# B&R Automation Studio project PLC code - cp (part 22)

#### Stack.st
```iecst
ACTION Stack:

	(* UA_MethodCall - call methode *)
	InputArguments_0[0].Name := 'MediaData';
	InputArguments_0[0].Value := '::SimMachFst:NewMediaData_0';
	OutputArguments_0[0].Name := 'Result';
	OutputArguments_0[0].Value := '::SimMachFst:MethodResult_0';
	UA_MethodCall_0(Execute := ExecuteMethodCall_0,
		ConnectionHdl := ConnectionHdl_0,
		MethodHdl := MethodHdl_0,
		Timeout := T#10s,
		InputArguments := InputArguments_0,
		OutputArguments := OutputArguments_0);
	IF NOT UA_MethodCall_0.Busy THEN
		ExecuteMethodCall_0 := FALSE;
		IF UA_MethodCall_0.Done THEN
			NewMediaData_0.rLength := NewMediaData_0.rLength + 1;
		END_IF
		IF UA_MethodCall_0.Error THEN
			NewMediaData_0.rDocLength := NewMediaData_0.rDocLength + 1;
		END_IF
	END_IF

	// Managing the automatic sending. Not sending if enable drying. Sendign Energy then
	IF NOT gThicknessCtrl.status.xNewMediaStackEnabled OR gThicknessCtrl.parameters.Dry.xDryStack THEN
		RETURN;
	END_IF

	IF (gSimMachine.Parameters.Stack.iMediaQuantityToKeepLoaded <= gThicknessCtrl.status.Stack.iNewMediaLoadedL1 + gThicknessCtrl.status.Stack.iNewMediaLoadedL2) THEN
		RETURN;
	END_IF

	// Adding a timer to avoid not working the method
	tonNotCallingMethod_0.IN := NOT UA_MethodCall_0.Busy;
	tonNotCallingMethod_0.PT := t#500ms;
	tonNotCallingMethod_0();
	IF EDGEPOS(tonNotCallingMethod_0.Q) THEN
		ExecuteMethodCall_0 := TRUE;
	END_IF

END_ACTION

ACTION InitialDataForMedia:

	NewMediaData_0.iLine := 1;
	NewMediaData_0.xHasWhite := FALSE;
	NewMediaData_0.rThickness := 3;
	NewMediaData_0.rWidth := 1400;
	NewMediaData_0.rLength := 1000;
	NewMediaData_0.rCrossOffset := 0;
	NewMediaData_0.rDocWidth := 1400;
	NewMediaData_0.rDocLength := 950;
	NewMediaData_0.rDocCrossOffset := 0;
	NewMediaData_0.rDocProcessOffset := 0;

END_ACTION

ACTION PreparingMethodComms:

	ExecuteConnect_0 := TRUE;

	(* UA_Connect - establish connection to OPC UA Server *)
	SessionConnectInfo_0.SecurityMsgMode := UASecurityMsgMode_None;
	SessionConnectInfo_0.SecurityPolicy := UASecurityPolicy_None;
	SessionConnectInfo_0.TransportProfile := UATP_UATcp;
	SessionConnectInfo_0.UserIdentityToken.UserIdentityTokenType := UAUITT_Username;
	SessionConnectInfo_0.UserIdentityToken.TokenParam1 := 'PressCore';
	SessionConnectInfo_0.UserIdentityToken.TokenParam2 := 'h98o76';
	SessionConnectInfo_0.SessionTimeout := T#1m;
	SessionConnectInfo_0.MonitorConnection := T#10s;

	UA_Connect_0(Execute := ExecuteConnect_0,
		ServerEndpointUrl := 'opc.tcp://localhost:4840',
	SessionConnectInfo := SessionConnectInfo_0,
	Timeout := T#10s);
	IF NOT UA_Connect_0.Busy THEN
		ExecuteConnect_0 := FALSE;
		IF UA_Connect_0.Done THEN
			ConnectionHdl_0 := UA_Connect_0.ConnectionHdl;
			////// NEXT
			ExecuteGetnamespaceindex_0 := TRUE;
		END_IF
		IF UA_Connect_0.Error THEN
			ConnectionHdl_0 := 0;
		END_IF
	END_IF

	(* UA_GetNamespaceIndex - read index of required namespace for PVs *)
	UA_GetNamespaceIndex_0(Execute := ExecuteGetnamespaceindex_0,
		ConnectionHdl := ConnectionHdl_0,
		NamespaceUri := 'http://br-automation.com/OpcUa/PLC/PV/',
	Timeout := T#5s);
	IF NOT UA_GetNamespaceIndex_0.Busy THEN
		ExecuteGetnamespaceindex_0 := FALSE;
		IF UA_GetNamespaceIndex_0.Done THEN
			NamespaceIndex_0 := UA_GetNamespaceIndex_0.NamespaceIndex;
			////// NEXT
			ExecuteMethodGetHandle_0 := TRUE;
		END_IF
		IF UA_GetNamespaceIndex_0.Error THEN
			NamespaceIndex_0 := 0;
		END_IF
	END_IF

	(* UA_MethodGetHandle - get a handle for required methode *)
	ObjectNodeID_0.NamespaceIndex := NamespaceIndex_0;
	ObjectNodeID_0.Identifier := '::ThickPos';
	ObjectNodeID_0.IdentifierType := UAIdentifierType_String;
	MethodNodeID_0.NamespaceIndex := NamespaceIndex_0;
	MethodNodeID_0.Identifier := '::ThickPos:LoadNewMedia';
	MethodNodeID_0.IdentifierType := UAIdentifierType_String;
	UA_MethodGetHandle_0(Execute := ExecuteMethodGetHandle_0,
		ConnectionHdl := ConnectionHdl_0,
		ObjectNodeID := ObjectNodeID_0,
		MethodNodeID := MethodNodeID_0,
		Timeout := T#10s);
	IF NOT UA_MethodGetHandle_0.Busy THEN
		ExecuteMethodGetHandle_0 := FALSE;
		IF UA_MethodGetHandle_0.Done THEN
			MethodHdl_0 := UA_MethodGetHandle_0.MethodHdl;
			////// NEXT
			// READY TO COMMUNICATE
		END_IF
		IF UA_MethodGetHandle_0.Error THEN
			MethodHdl_0 := 0;
		END_IF
	END_IF

END_ACTION
```

- Visualisation Logical/Printer/Sim/SimVisu (not shown)

### TestResources.var
```iecst
VAR
	iIndex : UDINT;
	iMax : UDINT;
	rVal : REAL;
END_VAR
```

- Visualisation Logical/Printer/mappView (not shown)

### Library Logical/UnitTest/Libraries/EFIAssert (ANSIC)

#### EFIAssert_ThresholdAssert.h - Threshold: macros
```c
/********************************************************************
 * COPYRIGHT -- Bernecker + Rainer
 ********************************************************************
 * Library: EFIAssert
 * File: EFIAssert_ThresholdAssert.h
 * Author: B+R
 *******************************************************************/

#include <bur/plctypes.h>

#include <bur/plctypes.h>
#include "UnitTest.h"

#ifdef __cplusplus
extern "C"
{
#endif

/* Dummies for smart edit autocompletion.
See below for the real macros used by the compiler  */
#ifdef _SMART_EDIT_DUMMY_
	/* This asserts checks (actual < threshold) */
	BOOL SPLEFI_ASSERT_UPPER_BOUNDARY(DINT threshold, DINT actual);
#endif

/*------------------------------------------------------------*/

/* Prototyping of functions.
These declaration of functions are used by the compiler to check number and type of arguments. */
BOOL splefi_assertUpperBoundary_DINT(const DINT threshold, const DINT actual, unsigned long line, const char *file);

/* Macros used in the test implementation.
The macro passes the location information to the implemented assert. */
#define SPLEFI_ASSERT_UPPER_BOUNDARY(threshold, actual) 	\
	splefi_assertUpperBoundary_DINT(threshold, actual, (unsigned long) __LINE__, __FILE__)

#ifdef __cplusplus
};
#endif
```

#### EFIAssert_REAL_ArrayAsserts.c - Array of REAL: implementation of the assert
```c
/********************************************************************
 * COPYRIGHT -- Bernecker + Rainer
 ********************************************************************
 * Library: EFIAssert
 * File: EFIAssert_REAL_ArrayAsserts.c
 * Author: B+R
 *******************************************************************/

#include <bur/plctypes.h>

#include "asbrstr.h"
#include "EFIAssert_REAL_ArrayAsserts.h"

#define TRUE 1
#define FALSE 0

#define NR_OF_DETAILED_ENTRIES_TO_SHOW 10

/* Tests each REAL in the array for equality in range
Returns true if passed, false otherwise
delta: allowed tolerance (floats are not exact values)
expected: array of expected REAL values
acutal: array of REAL values under test
nrOfEntries: number of entries in array
line: location information
file: location information
*/
BOOL splefi_assertImplRealArrayWithin(const REAL *delta,
                                   const REAL *expected, 	const REAL *actual, const unsigned long nrOfEntries,
                                   unsigned long line, const char *file)
{
	unsigned long i = 0;
	unsigned long countFail = 0;
	STRING buffer[100];
	STRING numbuf[30];

	/*------------------------------------------------------------*/
	for(i = 0; i < nrOfEntries; i++)
	{
		REAL diff = actual[i] - expected[i];
		REAL pos_delta = delta[i];

		if (diff < 0)
		{
			/* use absolute (positive) value */
			diff = 0.0f - diff;
		}
		if (pos_delta < 0)
		{
			/* use absolute (positive) value */
			pos_delta = 0.0f - pos_delta;
		}

		/* Check */
		if (pos_delta < diff)
		{
			/* count the failures */
			countFail++;

			/* for the first NR_OF_DETAILED_ENTRIES_TO_SHOW failures generate an informational message) */
			if(countFail < NR_OF_DETAILED_ENTRIES_TO_SHOW)
			{
				brsstrcpy((unsigned long) buffer, (unsigned long) "At array index ");
				brsitoa((int)i, (unsigned long)numbuf);
				brsstrcat((unsigned long) buffer, (unsigned long) numbuf);

				brsstrcat((unsigned long) buffer, (unsigned long) ": exp ");
				brsftoa((REAL)expected[i], (unsigned long)numbuf);
				brsstrcat((unsigned long) buffer, (unsigned long) numbuf);

				brsstrcat((unsigned long) buffer, (unsigned long)" was ");
				brsftoa((REAL)actual[i], (unsigned long)numbuf);
				brsstrcat((unsigned long) buffer, (unsigned long) numbuf);

				addInfo(buffer, line, file);
			}
		}
	}/* end for */
	/*------------------------------------------------------------*/
	/* All entries checked, generate notification for test report */
	if(0 == countFail)
	{
		addPassed("", line, file);
		return TRUE;
	}
	else
	{
		brsitoa(countFail, (unsigned long)numbuf);
		brsstrcpy((unsigned long)buffer, (unsigned long)numbuf);
		brsstrcat((unsigned long)buffer, (unsigned long)" failures occured in array ");
		addFailure(buffer, line, file);
		return FALSE;
	}
}

/* Tests each REAL in the array for equality
Returns true if passed, false otherwise
delta: allowed tolerance (floats are not exact values)
expected: array of expected REAL values
acutal: array of REAL values under test
nrOfEntries: number of entries in array
line: location information
file: location information
*/
BOOL splefi_assertImplRealArrayEqual(const REAL delta,
                                  const REAL *expected, 	const REAL *actual, const unsigned long nrOfEntries,
                                  unsigned long line, const char *file)
{
	unsigned long i = 0;
	char countFail = 0;
	STRING buffer[100];
	STRING numbuf[30];

	/*------------------------------------------------------------*/
	for(i = 0; i < nrOfEntries; i++)
	{
		REAL diff = actual[i] - expected[i];
		REAL pos_delta = delta * (REAL)(expected[i]);

		if (diff < 0)
		{
			/* use absolute (positive) value */
			diff = 0.0f - diff;
		}
		if (pos_delta < 0)
		{
			/* use absolute (positive) value */
			pos_delta = 0.0f - pos_delta;
		}

		/* Check */
		if (pos_delta < diff)
		{
			/* count the failures */
			countFail++;

			/* for the first NR_OF_DETAILED_ENTRIES_TO_SHOW failures generate an informational message) */
			if(countFail < NR_OF_DETAILED_ENTRIES_TO_SHOW)
			{
				brsstrcpy((unsigned long) buffer, (unsigned long) "At array index ");
				brsitoa((int)i, (unsigned long) numbuf);
				brsstrcat((unsigned long) buffer, (unsigned long) numbuf);

				brsstrcat((unsigned long) buffer, (unsigned long) ": exp ");
				brsftoa((REAL)expected[i], (unsigned long)numbuf);
				brsstrcat((unsigned long) buffer, (unsigned long) numbuf);

				brsstrcat((unsigned long) buffer, (unsigned long) " was ");
				brsftoa((REAL)actual[i], (unsigned long)numbuf);
				brsstrcat((unsigned long) buffer, (unsigned long) numbuf);

				addInfo(buffer, 0, 0);
			}
		}
	}/* end for */

	/*------------------------------------------------------------*/
	/* All entries checked, generate notification for test report */
	if(0 == countFail)
	{
		addPassed("", line, file);
		return TRUE;
	}
	else
	{
		brsitoa(countFail, (unsigned long)numbuf);
		brsstrcpy((unsigned long)buffer, (unsigned long)numbuf);
		brsstrcat((unsigned long)buffer,(unsigned long) " failures occured in array ");
		addFailure(buffer, line, file);
		return FALSE;
	}
}
```

#### EFIAssert_GreaterThanReal.c - GreaterThanReal: implementation of the assert
```c
#include <bur/plctypes.h>

#include "asbrstr.h"
#include "EFIAssert_GreaterThanReal.h"

#define TRUE 1
#define FALSE 0

/* Returns TRUE if assert passed; FALSE otherwise
	function variables
	threshold: minimum accepted value
	actual: test value
	line: location information
	file: location information
*/

BOOL efi_assertGreaterThanReal_REAL (const REAL threshold, const REAL actual, const long line, const char *file){
	STRING buffer[100];
	STRING numbuf[16];

	//conditions
	if(threshold < actual){
		//passed assert
		addPassed("", line, file);
		return TRUE;
	}
	else{
		//failed assert

		//error message
		brsstrcpy((unsigned long) buffer, (unsigned long) "Limit of ");
		brsftoa((float)threshold, (unsigned long) numbuf);
		brsstrcat((unsigned long) buffer, (unsigned long) numbuf);
		brsstrcat((unsigned long) buffer, (unsigned long) " was exceded. Actual was ");

		brsftoa((float)actual, (unsigned long) numbuf);
		brsstrcat((unsigned long) buffer, (unsigned long) numbuf);
		brsstrcat((unsigned long) buffer, (unsigned long) ".");

		//failure report
		addFailure(buffer, line, file);
		return FALSE;

	}
};
```

#### EFIAssert_GreaterThanReal.h - GreaterThanReal: macros
```c
#include <bur/plctypes.h>

#include <bur/plctypes.h>
#include "UnitTest.h"

#ifdef __cplusplus
extern "C"
{
#endif

// Dummies for smartedit
#ifdef _SMART_EDIT_DUMMY_
	/* This asserts checks (actual < threshold) */
	BOOL EFI_ASSERT_GREATER_THAN_REAL(REAL threshold, REAL actual);
#endif

// Prototypes
	BOOL efi_assertGreaterThanReal_REAL (const REAL threshold,const REAL actual, const long line, const char *file);

// Macros
#define EFI_ASSERT_GREATER_THAN_REAL(threshold, actual) 	\
	efi_assertGreaterThanReal_REAL(threshold, actual, (unsigned long) __LINE__, __FILE__)

#ifdef __cplusplus
};
#endif
```

### Program Logical/UnitTest/Libraries/LibAssert1

#### LibAssert1.h
```c
/********************************************************************
 * COPYRIGHT -- Bernecker + Rainer
 ********************************************************************
 * Library: LibAssert1
 * File: LibAssert1.h
 * Author: B+R
 *******************************************************************/

#include <bur/plctypes.h>
#include "UnitTest.h"

/* When this file is included the defines, makros  of the following header files should be provided as well:  */

#include "LibAssert1_REAL_ArrayAsserts.h"
#include "LibAssert1_ThresholdAssert.h"
```

#### LibAssert1_REAL_ArrayAsserts.h
```c
/********************************************************************
 * COPYRIGHT -- Bernecker + Rainer
 ********************************************************************
 * Library: LibAssert1
 * File: LibAssert1_REAL_ArrayAsserts.h
 * Author: B+R
 *******************************************************************/

#include <bur/plctypes.h>
#include "UnitTest.h"

#ifdef __cplusplus
extern "C"
{
#endif

	/* Dummies for smart edit autocompletion.
	See below for the real macros used by the compiler  */
#ifdef _SMART_EDIT_DUMMY_

	/* This assert checks two arrays of floats for equality. TEST_FLOAT_PRECISION is used as default Delta.

	Note: An assert like this is generally more readable and meaningful than multiple TEST_ASSERT_EQUAL_FLOAT().
	It informs about how many entries failed in total and shows the first NR_OF_DETAILED_ENTRIES_TO_SHOW together with the array index the failure occured. */
	BOOL SPL_ASSERT_ARRAY_EQUAL_REAL(REAL *expected[], REAL *actual[], UDINT nrOfEntries);

	/* This assert checks two arrays of floats for equality with an accepted delta per entry

	Note: An assert like this is generally more readable and meaningful than multiple TEST_ASSERT_FLOAT_WITHIN().
	It informs about how many entries failed in total and shows the first NR_OF_DETAILED_ENTRIES_TO_SHOW together with the array index the failure occured.
	*/
	BOOL SPL_ASSERT_ARRAY_REAL_WITHIN(REAL *delta[], REAL *expected[], REAL *actual[], UDINT nrOfEntries);

#endif

	/*------------------------------------------------------------*/

	/* Prototyping of functions.
	These declaration of functions are used by the compiler to check number and type of arguments. */
	BOOL spl_assertImplRealArrayEqual(const REAL delta,
	                                  const REAL *expected,
	                                  const REAL *actual,
	                                  const unsigned long nrOfEntries,
	                                  unsigned long line, const char *file);

	BOOL spl_assertImplRealArrayWithin(const REAL *delta,
	                                   const REAL *expected,
	                                   const REAL *actual,
	                                   const unsigned long nrOfEntries,
	                                   unsigned long line, const char *file);

	/* Makros used in the test implementation.
	The macro passes the location information to the implemented assert. */

#define SPL_ASSERT_ARRAY_EQUAL_REAL(expected, actual, nrOfEntries)	\
	spl_assertImplRealArrayEqual((REAL)TEST_FLOAT_PRECISION, expected, actual, nrOfEntries, (unsigned long) __LINE__, __FILE__)

#define SPL_ASSERT_ARRAY_REAL_WITHIN(delta, expected, actual, nrOfEntries)	\
	spl_assertImplRealArrayWithin(delta, expected, actual, nrOfEntries,  (unsigned long) __LINE__, __FILE__)

#ifdef __cplusplus
};
#endif
```

#### LibAssert1_ThresholdAssert.h
```c
/********************************************************************
 * COPYRIGHT -- Bernecker + Rainer
 ********************************************************************
 * Library: LibAssert1
 * File: LibAssert1_ThresholdAssert.h
 * Author: B+R
 *******************************************************************/

#include <bur/plctypes.h>

#include <bur/plctypes.h>
#include "UnitTest.h"

#ifdef __cplusplus
extern "C"
{
#endif

/* Dummies for smart edit autocompletion.
See below for the real macros used by the compiler  */
#ifdef _SMART_EDIT_DUMMY_
	/* This asserts checks (actual < threshold) */
	BOOL SPL_ASSERT_UPPER_BOUNDARY(DINT threshold, DINT actual);
#endif

/*------------------------------------------------------------*/

/* Prototyping of functions.
These declaration of functions are used by the compiler to check number and type of arguments. */
BOOL spl_assertUpperBoundary_DINT(const DINT threshold, const DINT actual, unsigned long line, const char *file);

/* Macros used in the test implementation.
The macro passes the location information to the implemented assert. */
#define SPL_ASSERT_UPPER_BOUNDARY(threshold, actual) 	\
	spl_assertUpperBoundary_DINT(threshold, actual, (unsigned long) __LINE__, __FILE__)

#ifdef __cplusplus
};
#endif
```

#### LibAssert1_ThresholdAssert.c
```c
/********************************************************************
 * COPYRIGHT -- Bernecker + Rainer
 ********************************************************************
 * Library: LibAssert1
 * File: LibAssert1_ThresholdAssert.c
 * Author: B+R
 *******************************************************************/

#include <bur/plctypes.h>

#include "asbrstr.h"
#include "LibAssert1_ThresholdAssert.h"

#define TRUE 1
#define FALSE 0

/* Returns TRUE: Assert passed, FALSE otherwise
threshold: limit
actual: value under test
line: location information
file: location information
*/
BOOL spl_assertUpperBoundary_DINT(const DINT threshold, const DINT actual,
                                  unsigned long line, const char *file)
{
	STRING buffer[100];
	STRING numbuf[15];

	/* Check */
	if(threshold > actual) /* Good case: actual value is below the allowed (expected) maximum. */
	{
		/* Inform the test framework about a passed assert*/
		addPassed("", line, file);
		return TRUE;
	}
	else /* Bad case: acutal value exceeded acceptable threshold  */
	{
		/* Generate message for failure */
		brsstrcpy((unsigned long) buffer, (unsigned long) "Limit ");
		brsitoa((int)threshold, (unsigned long)numbuf);
		brsstrcat((unsigned long) buffer, (unsigned long) numbuf);
		brsstrcat((unsigned long) buffer, (unsigned long) " exceeded (was ");

		brsitoa((int)actual, (unsigned long)numbuf);
		brsstrcat((unsigned long) buffer, (unsigned long) numbuf);
		brsstrcat((unsigned long) buffer, (unsigned long) " ) ");

		/* Add failure to test report */
		addFailure(buffer, line, file);
		return FALSE;
	}
};
```

### UnitTest.h
```c
/*****************************************************************************
 * COPYRIGHT (C) BERNECKER + RAINER
 *****************************************************************************
 * Library:  UnitTest
 * File:     UnitTest.h
 * Author:   B+R
 *****************************************************************************
 * Description: Static library for UnitTest programs written in ANSI C /C++
 *
 * Add the path "\Logical\TS_UnitTest\Libraries\UnitTest\" to the
 * "Additional include directories" in the tab "Build" (PLC Properties)
 ******************************************************************************/

#ifndef	__UNITTEST_H__
#define	__UNITTEST_H__
#ifdef __cplusplus
extern "C"
{
#endif
#include <bur/plctypes.h>

#ifndef NULL
#define	NULL	0
#endif
#include "include/Test.h"

#include "include/TestCase.h"
#include "include/TestListener.h"
#include "include/TestResult.h"
#include "include/TestCaller.h"

#include "include/AssertImpl.h"
#include "include/HelperMacro.h"
#include "include/utRunner.h"

/* function is a test case */
#define _TEST 			static testStatusEnum

/* function is a setup */
#define _SETUP_TEST 	static testStatusEnum 	setupTest

/* function is a teardown */
#define _TEARDOWN_TEST 	static testStatusEnum 	teardownTest

/* function is a setup for whole test set */
#define _SETUP_SET		static testStatusEnum	setupSet

/* function is a teardown for whole test set */
#define _TEARDOWN_SET 	static testStatusEnum	teardownSet

/* function is a cyclic handler for test set */
#define _CYCLIC_SET		static void 			cyclicSetCaller

/* Skipped test case */
#define SKIP_TEST  		_TEST
/* Skip all test cases of set */
#define SKIP_TEST_SET

/* Dummies for smart edit autocompletion.
See AssertImpl.h for real macros used by the compiler  */
#ifdef _SMART_EDIT_DUMMY_

/* String comparison.
Returns true if the strings are equal. */
BOOL TEST_ASSERT_EQUAL_STRING(char *expected,char  *actual);
/* Wstring comparison.
Returns true if the WSTRINGS are equal. */
BOOL TEST_ASSERT_EQUAL_WSTRING(unsigned short *expected,unsigned short *actual);
 /* Compares two memory blocks.
Returns true if [size] bytes are equal. */
BOOL TEST_ASSERT_EQUAL_MEM(void *expected, void *actual,UDINT size);
/* Compares integer values. Usable for all integer types.
Avoid comparison of unsigned with signed types.
Returns true if they are equal.
Note: If different, values are reported as DINT values in the test report */
BOOL TEST_ASSERT_EQUAL_INT(expected, actual);

/* Compares REAL values with delta = (expected * TEST_FLOAT_PRECISION).
Returns true if (difference <= delta) */
BOOL TEST_ASSERT_EQUAL_REAL(REAL expected,REAL actual);
/* Compares REAL values with explicit delta.
Returns true if (difference <= delta) */
BOOL TEST_ASSERT_REAL_WITHIN(REAL delta, REAL expected, REAL actual);
/* Compares LREAL values with delta = (expected * TEST_DOUBLE_PRECISION).
Returns true if (difference <= delta) */
BOOL TEST_ASSERT_EQUAL_LREAL(LREAL expected,LREAL  actual);
/* Compares LREAL values with explicit delta.
Returns true if (difference <= delta) */
BOOL TEST_ASSERT_LREAL_WITHIN(LREAL delta, LREAL expected, LREAL actual);

/* Compares float values with delta = (expected * TEST_FLOAT_PRECISION).
Returns true if (difference <= delta) */
BOOL TEST_ASSERT_EQUAL_FLOAT(float expected, float actual);
/* Compares float values with explicit delta.
Returns true if (difference <= delta) */
BOOL TEST_ASSERT_FLOAT_WITHIN(float delta, float expected, float actual);
/* Compares double values with delta = (expected * TEST_DOUBLE_PRECISION).
Returns true if (difference <= delta) */
BOOL TEST_ASSERT_EQUAL_DOUBLE(double expected, double actual);
/* Compares double values with explicit delta.
Returns true if (difference <= delta) */
BOOL TEST_ASSERT_DOUBLE_WITHIN(double delta, double expected, double actual);

/* Returns true if pointer is null */
BOOL TEST_ASSERT_NULL(void *pointer);
/* Returns true if pointer is not null */
BOOL TEST_ASSERT_NOT_NULL(void *pointer);
/* Returns true, if condition evals to  true */
BOOL TEST_ASSERT_MESSAGE(condition, char *message);
/* Returns true, if condition evals to  true */
BOOL TEST_ASSERT(condition);

/* Returns always false */
BOOL TEST_FAIL(char *message);

/* Add a note to the test report */
void TEST_INFO(char *message);
/* Add a note with location information to the test report */
void TEST_INFO_POS(char *message);

#ifdef __cplusplus
/* Test if expression throws given exception.
Catches all other exceptions as failure.
Note: Available for C++ only */
void TEST_ASSERT_THROW(expression, type);

/* Fails if expression throws any exceptions.
Note: Available for C++ only*/
void TEST_ASSERT_NO_THROW(expression);
#endif

/* Adds a test function with description to the Testfixture.
See UNITTEST_FIXTURES() */
void new_TestFixture(char *name, _TEST function);

/* Adds a test function with description to the Testfixture.
This test will be skipped
See UNITTEST_FIXTURES() */
void skipTestFixture(char *name, _TEST function);

/* Defines the order of test cases.
Should look like this
UNITTEST_FIXTURES(fixtures)
{
	new_TestFixture("test_1",test_1),
	new_TestFixture("test_2",test_2),
	new_TestFixture("test_3",test_3)
}
*/
void UNITTEST_FIXTURES(fixtures)

/* Standard UnitTest caller without any setup / teardown methods*/
void UNITTEST_CALLER_TEST(caller, char *name, fixtures);

/* Standard UnitTest caller with macro setup / teardown for tests*/
void UNITTEST_CALLER_BASIC(caller, char *name, fixtures);

/* UnitTest caller with macro setup / teardown for tests and test set */
void UNITTEST_CALLER_SET(caller, char *name, fixtures);

/* UnitTest caller with macro setup / teardown for tests and test set and cylic*/
void UNITTEST_CALLER_COMPLETE(caller, char *name, fixtures);

/* UnitTest caller with explicit setup / teardown for suite */
void UNITTEST_CALLER_SET_EXPLICIT(caller,name,setupTest,teardownTest,fixtures, setupSuite, teardownSuite);

/* UnitTest caller with explicit setup / teardown for suite and cylic */
void UNITTEST_CALLER_COMPLETE_EXPLICIT(caller,name,setupTest,teardownTest,fixtures, setupSuite, teardownSuite, cyclicCaller);

/* Adds a test set with description to the fixture of test sets.
See UNITTEST_TESTSET_FIXTURES() */
void new_TestSet(testcaller);

/* Defines the order of test sets.
Should look like this
UNITTEST_TESTSET_FIXTURES(fixtures)
{
	new_TestSet(testSet_1),
	new_TestSet(testSet_2),
	new_TestSet(testSet_3)
}*/
void UNITTEST_TESTSET_FIXTURES(fixtures);

/* Defines the test set list handling structure*/
void UNTITTEST_TESTSET_HANDLER();

#endif /*_SMART_EDIT_DUMMY_*/

/*
 Use to declare Test set for use in list of test sets of test programm
 See usage in autogeneratedFile.c / FixtureOfTestSets.c
*/
#define UNITTEST_TESTSET_DECLARATION 	extern const TestCaller

/* Default factor for precision used to test if REAL / float values  are equal.
(0.00001f) */
#define TEST_FLOAT_PRECISION 	(0.00001f)
/* Default factor for precision used to test if LREAL / double values  are equal.
(1e - 12f) */
#define TEST_DOUBLE_PRECISION 	(1e-12f)

#if (__GNUC__ != 4) || (__GNUC_MINOR__ != 1) || (__GNUC_PATCHLEVEL__ != 2)
#warning UnitTest is compiled with GCC version 4.1.2. To use UnitTest switch GCC version to 4.1.2 or use different solution package
#endif

#define UNIT_TEST_LIBRARY_VERSION  			"2.01.0"

#ifdef __cplusplus
};
#endif

#include "include/asserts.hpp"

#endif/*__UNITTEST_H__*/
```

### AssertImpl.h - Available asserts
```c
/*
* Author: 		B+R
* Contents of this file are modified and extended
*/

/*
 * COPYRIGHT AND PERMISSION NOTICE
 *
 * Copyright (c) 2003 Embedded Unit Project
 *
 * All rights reserved.
 *
 * Permission is hereby granted, free of charge, to any person obtaining
 * a copy of this software and associated documentation files (the
 * "Software"), to deal in the Software without restriction, including
 * without limitation the rights to use, copy, modify, merge, publish,
 * distribute, and/or sell copies of the Software, and to permit persons
 * to whom the Software is furnished to do so, provided that the above
 * copyright notice(s) and this permission notice appear in all copies
 * of the Software and that both the above copyright notice(s) and this
 * permission notice appear in supporting documentation.
 *
 * THE SOFTWARE IS PROVIDED "AS IS", WITHOUT WARRANTY OF ANY KIND,
 * EXPRESS OR IMPLIED, INCLUDING BUT NOT LIMITED TO THE WARRANTIES OF
 * MERCHANTABILITY, FITNESS FOR A PARTICULAR PURPOSE AND NONINFRINGEMENT
 * OF THIRD PARTY RIGHTS. IN NO EVENT SHALL THE COPYRIGHT HOLDER OR
 * HOLDERS INCLUDED IN THIS NOTICE BE LIABLE FOR ANY CLAIM, OR ANY
 * SPECIAL INDIRECT OR CONSEQUENTIAL DAMAGES, OR ANY DAMAGES WHATSOEVER
 * RESULTING FROM LOSS OF USE, DATA OR PROFITS, WHETHER IN AN ACTION OF
 * CONTRACT, NEGLIGENCE OR OTHER TORTIOUS ACTION, ARISING OUT OF OR IN
 * CONNECTION WITH THE USE OR PERFORMANCE OF THIS SOFTWARE.
 *
 * Except as contained in this notice, the name of a copyright holder
 * shall not be used in advertising or otherwise to promote the sale,
 * use or other dealings in this Software without prior written
 * authorization of the copyright holder.
 *
 * $Id: AssertImpl.h,v 1.6 2003/09/16 11:09:53 arms22 Exp $
 */

#ifndef	__ASSERTIMPL_H__
#define	__ASSERTIMPL_H__

#ifdef	__cplusplus
extern "C" {
#endif

#include <bur/plctypes.h>

/* Increments failure counter and outputs failure text*/
void addFailure(const char *msg, unsigned long line, const char *file);
/* Increments passed counter*/
void addPassed(const char *msg, unsigned long line, const char *file);
/* Outputs informational text*/
void addInfo(const char *msg, unsigned long line, const char *file);
/* Increments abort counter, aborts current test set, outputs abort text.
    Existing teardown methods will be called before leaving the test set */
void addAbort(const char *msg, unsigned long line, const char *file);

BOOL assertImplementationInt(int expected,int actual, unsigned long line, const char *file);
BOOL assertImplementationCStr(const char *expected,const char *actual, unsigned long line, const char *file);
BOOL assertImplementationDoublesWithin(const double delta,	const double expected,	const double actual,	unsigned long line, const char *file);
BOOL assertImplementationFloatsWithin(const float delta,	const float expected,	const float actual,	unsigned long line, const char *file);
BOOL assertImplementationWStr(const unsigned short *expected,const unsigned short *actual, unsigned long line, const char *file);
BOOL assertCondition(BOOL condition, const char *message,  unsigned long line, const char *file);
BOOL assertImplementationMem(void *expected ,void  *actual, unsigned long  size, unsigned long line, const char *file);

#define TEST_ASSERT_EQUAL_STRING(expected,actual)\
	assertImplementationCStr(expected,actual,__LINE__,__FILE__)

#define TEST_ASSERT_EQUAL_WSTRING(expected,actual)\
	assertImplementationWStr(expected,actual,__LINE__,__FILE__)

#define TEST_ASSERT_EQUAL_MEM(expected,actual,size)\
	assertImplementationMem(expected,actual,size,__LINE__,__FILE__)

#define TEST_ASSERT_EQUAL_INT(expected,actual)\
	assertImplementationInt(expected, actual,__LINE__,__FILE__)

#define TEST_ASSERT_NULL(pointer)\
	TEST_ASSERT_MESSAGE(pointer == NULL,#pointer " was not null.")

#define TEST_ASSERT_NOT_NULL(pointer)\
	TEST_ASSERT_MESSAGE(pointer != NULL,#pointer " was null.")

#define TEST_ASSERT_MESSAGE(condition, message)\
	assertCondition(condition,message,__LINE__,__FILE__)

#define TEST_ASSERT(condition) \
	assertCondition(condition, #condition,__LINE__,__FILE__)

#define TEST_FAIL(message)\
	assertCondition(0, message,__LINE__,__FILE__)

#define TEST_ASSERT_EQUAL_FLOAT(expected, actual)   		\
	assertImplementationFloatsWithin(\
									 (float)(expected) * (float)TEST_FLOAT_PRECISION, \
									 (float)(expected), (float)(actual), \
									 (unsigned long) __LINE__, __FILE__)

#define TEST_ASSERT_FLOAT_WITHIN(delta, expected, actual)	 \
	assertImplementationFloatsWithin(\
									 (float)(delta), \
									 (float)(expected), (float)(actual), \
									 (unsigned long) __LINE__, __FILE__)

#define TEST_ASSERT_EQUAL_DOUBLE(expected, actual)           \
	assertImplementationDoublesWithin(\
									  (double)(expected) * (double)TEST_DOUBLE_PRECISION,\
									  (double)(expected), (double)(actual), \
									  (unsigned long) __LINE__, __FILE__)

#define TEST_ASSERT_DOUBLE_WITHIN(delta, expected, actual)    \
	assertImplementationDoublesWithin(\
									  (double)(delta),\
									  (double)(expected), (double)(actual), \
									  (unsigned long) __LINE__, __FILE__)

	/* IEC data types*/
#define TEST_ASSERT_EQUAL_REAL(expected, actual)     		TEST_ASSERT_EQUAL_FLOAT(expected, actual)
#define TEST_ASSERT_REAL_WITHIN(delta, expected, actual)    TEST_ASSERT_FLOAT_WITHIN(delta, expected, actual)

#define TEST_ASSERT_EQUAL_LREAL(expected, actual)  			TEST_ASSERT_EQUAL_DOUBLE(expected, actual)
#define TEST_ASSERT_LREAL_WITHIN(delta, expected, actual)	TEST_ASSERT_DOUBLE_WITHIN(delta, expected, actual)

#define TEST_INFO(message)		addInfo(message,0,0);
#define TEST_INFO_POS(message)	addInfo(message,__LINE__,__FILE__)

	/* Returns and signals completion.
	Note: This is a return statement*/
#define TEST_DONE 				return ut_DONE

	/* Returns and signals that this call is not yet completed. Will be called again in next cycle.
	Note: This is a conditional return statement*/
#define TEST_BUSY 				return ut_BUSY

	/* If condition is true: Returns and signals that this call is not yet completed. Will be called again in next cycle.
	Note: This is a conditional return statement */
#define TEST_BUSY_CONDITION(condition) 				if(condition) { 	TEST_BUSY; }
	/* If condition is true: Returns and signals that this call is not yet completed. Will be called again in next cycle.
	A message is reported.
	Note: This is a conditional return statement*/
#define TEST_BUSY_CONDITION_MSG(condition, msg) 	if(condition) {	TEST_INFO( msg );  TEST_BUSY; }

	/* Returns and signals abortion of current test set.
	No further test case of this set will be executed.
	If available teardown methods will be called before test set is left.
	Note: This is a return statement*/
#define TEST_ABORT								{addAbort("Test set aborted.",__LINE__,__FILE__);} return ut_ABORT

	/* Returns and signals that this test case is aborted.
	No further test case of this set will be executed.
	If available teardown methods will be called before test set is left.
	A message is reported.
	Note: This is a return statement*/
#define TEST_ABORT_MSG(message)					{addAbort(message,__LINE__,__FILE__);} return ut_ABORT

	/* If condition is true: Returns and signals that this test case is aborted.
	No further test case of this set will be executed.
	If available teardown methods will be called before test set is left.
	Note: This is a conditional return statement*/
#define TEST_ABORT_CONDITION(condition) 				if(condition) { 	TEST_ABORT; }

	/* If condition is true: Returns and signals that this test case is aborted.
	No further test case of this set will be executed.
	If available teardown methods will be called before test set is left.
	A message is reported
	Note: This is a conditional return statement*/
#define TEST_ABORT_CONDITION_MSG(condition, msg) 		if(condition) { TEST_ABORT_MSG(msg); }

#ifdef	__cplusplus
}
#endif

#endif/*__ASSERTIMPL_H__*/
```

### Asserts.hpp
```cpp
/*****************************************************************************
 * COPYRIGHT (C) BERNECKER + RAINER
 *****************************************************************************
 * Library:  UnitTest
 * File:     Asserts.hpp
 * Author:   B+R
 ******************************************************************************/

#include <bur/plctypes.h>

#ifdef __cplusplus

#ifndef	__ASSERTIMPL_CPP_H__
#define	__ASSERTIMPL_CPP_H__

#include <string>

#define TEST_ASSERT_THROW(expression, type  ) \
		do { bool succeeded = false; std::string message( "Expected exception: " #type " not thrown."); \
		try {  expression;  }\
		catch ( const type & ) { succeeded = true;}\
		catch ( const std::exception &e ) { if(!succeeded) { message = "Unexpected exception caught: "; message += e.what();  message += ". Expected: "  #type;  }  }\
		catch ( ... ) { if(!succeeded) { message = "Unexpected exception caught. Expected: "   #type;  }  } \
		if ( succeeded  )  { addPassed("", __LINE__, __FILE__); } \
		else {   addFailure(message.c_str(), __LINE__, __FILE__ ); } \
		} while ( false )

#define TEST_ASSERT_NO_THROW(expression  ) \
		do { bool succeeded = false; 	std::string message(""); \
		try {  expression; succeeded = true;  } \
		catch ( const std::exception &e ) {message += ("Unexpected exception caught: " );  message +=  e.what(); }  \
		catch ( ... ) { message +=  "Unexpected exception caught."; }\
		if ( succeeded  )  { addPassed("", __LINE__, __FILE__); } \
		else { addFailure(message.c_str(), __LINE__, __FILE__ );}  \
		} while ( false )

#define TEST_ASSERT_EQUAL_OBJ(expected,actual)		 assertEquals((expected), (actual),  (UDINT)__LINE__, (const char*) __FILE__);

template <class T>
struct assertion__toString_typ
{
	static std::string toString( const T& x )
	{
		return x.c_str();
	}
};

template <class T>
bool assertEquals( const T& expected, const T& actual, unsigned long line, const char *file )
{
	if ( (expected == actual) )
	{
		addPassed("", line, file);
		return true;
	}
	else
	{
		std::string tmp("Objects are not equal. Expected \"");
		tmp += expected.toString()+ "\" was: \""  + actual.toString() + "\"";
		addFailure(tmp.c_str(), line, file);
		return false;
	}
}

#endif /* __ASSERTIMPL_CPP_H__*/

#endif
```

### HelperMacro.h
```c
/*
* Author: 		B+R
* Contents of this file are modified and extended
*/

/*
 * COPYRIGHT AND PERMISSION NOTICE
 *
 * Copyright (c) 2003 Embedded Unit Project
 *
 * All rights reserved.
 *
 * Permission is hereby granted, free of charge, to any person obtaining
 * a copy of this software and associated documentation files (the
 * "Software"), to deal in the Software without restriction, including
 * without limitation the rights to use, copy, modify, merge, publish,
 * distribute, and/or sell copies of the Software, and to permit persons
 * to whom the Software is furnished to do so, provided that the above
 * copyright notice(s) and this permission notice appear in all copies
 * of the Software and that both the above copyright notice(s) and this
 * permission notice appear in supporting documentation.
 *
 * THE SOFTWARE IS PROVIDED "AS IS", WITHOUT WARRANTY OF ANY KIND,
 * EXPRESS OR IMPLIED, INCLUDING BUT NOT LIMITED TO THE WARRANTIES OF
 * MERCHANTABILITY, FITNESS FOR A PARTICULAR PURPOSE AND NONINFRINGEMENT
 * OF THIRD PARTY RIGHTS. IN NO EVENT SHALL THE COPYRIGHT HOLDER OR
 * HOLDERS INCLUDED IN THIS NOTICE BE LIABLE FOR ANY CLAIM, OR ANY
 * SPECIAL INDIRECT OR CONSEQUENTIAL DAMAGES, OR ANY DAMAGES WHATSOEVER
 * RESULTING FROM LOSS OF USE, DATA OR PROFITS, WHETHER IN AN ACTION OF
 * CONTRACT, NEGLIGENCE OR OTHER TORTIOUS ACTION, ARISING OUT OF OR IN
 * CONNECTION WITH THE USE OR PERFORMANCE OF THIS SOFTWARE.
 *
 * Except as contained in this notice, the name of a copyright holder
 * shall not be used in advertising or otherwise to promote the sale,
 * use or other dealings in this Software without prior written
 * authorization of the copyright holder.
 *
 * $Id: HelperMacro.h,v 1.3 2004/02/10 16:19:29 arms22 Exp $
 */

#ifndef	__HELPERMACRO_H__
#define	__HELPERMACRO_H__

/* Defines the order of test cases */
#define UNITTEST_FIXTURES(fixtures) \
	static const TestFixture	fixtures[] =

/* Standard UnitTest caller without any setup / teardown methods*/
#define UNITTEST_CALLER_TEST(caller,name,fixtures) \
	UNITTEST_CALLER_COMPLETE_EXPLICIT(caller,name,0,0,fixtures,0,0, 0)

/* Standard UnitTest caller with macro setup / teardown for tests*/
#define UNITTEST_CALLER_BASIC(caller,name,fixtures) \
	UNITTEST_CALLER_COMPLETE_EXPLICIT(caller,name,setupTest,teardownTest,fixtures,0,0, 0)

/* UnitTest caller with macro setup / teardown for tests and test set */
#define UNITTEST_CALLER_SET(caller,name,fixtures) \
	UNITTEST_CALLER_COMPLETE_EXPLICIT(caller,name,setupTest,teardownTest,fixtures, setupSet, teardownSet, 0)

/* UnitTest caller with macro setup / teardown for tests and test set and cylic*/
#define UNITTEST_CALLER_COMPLETE(caller,name,fixtures) \
	UNITTEST_CALLER_COMPLETE_EXPLICIT(caller,name,setupTest,teardownTest,fixtures, setupSet, teardownSet, cyclicSetCaller)

/* UnitTest caller with explicit setup / teardown for suite */
#define UNITTEST_CALLER_SET_EXPLICIT(caller,name,sup,tdw,fixtures, setupSuite, teardownSuite) \
	UNITTEST_CALLER_COMPLETE_EXPLICIT(caller,name,sup,tdw,fixtures, setupSuite, teardownSuite, 0)

#ifdef  __cplusplus
/* UnitTest caller with explicit setup / teardown for suite and cylic */
#define UNITTEST_CALLER_COMPLETE_EXPLICIT(caller,name,sup,tdw,fixtures, setupSuite, teardownSuite, cyclicCaller) \
	UNITTEST_TESTSET_DECLARATION caller = new_TestCaller(name,sup,tdw,sizeof(fixtures)/sizeof(fixtures[0]),(TestFixture*)fixtures, setupSuite, teardownSuite, cyclicCaller)

#else

/* UnitTest caller with explicit setup / teardown for suite and cylic */
#define UNITTEST_CALLER_COMPLETE_EXPLICIT(caller,name,sup,tdw,fixtures, setupSuite, teardownSuite, cyclicCaller) \
	 const TestCaller caller = new_TestCaller(name,sup,tdw,sizeof(fixtures)/sizeof(fixtures[0]),(TestFixture*)fixtures, setupSuite, teardownSuite, cyclicCaller)

#endif

#define UNITTEST_CALLER_SKIPPED(caller,name,sup,tdw,fixtures, setupSuite, teardownSuite, cyclicCaller) \
 const TestCaller caller = skipTestCaller(name,sup,tdw,sizeof(fixtures)/sizeof(fixtures[0]),(TestFixture*)fixtures, setupSuite, teardownSuite, cyclicCaller)

/* --------------------------------------*/

/* --------------------------------------*/

typedef struct TestSetActive
{
	BOOL			active;
	TestCallerRef 	set;
} TestSetActive;

typedef struct TestSetList
{
	UINT 			nrOfTestSets;
	UINT 			currentTestSet;
	TestSetActive 	*list;
} TestSetList;

/* Defines the order of test sets.
Should look like this
UNITTEST_TESTSET_FIXTURES(fixtures)
{
	new_TestSet(testSet_1),
	new_TestSet(testSet_2),
	new_TestSet(testSet_3)
}*/
#define UNITTEST_TESTSET_FIXTURES(fixtures) \
	static TestSetActive	fixtures[] =

/* Adds a test set with description to the fixture of test sets.
See UNITTEST_TESTSET_FIXTURES() */
#define new_TestSet(testcaller)\
	{\
		1,\
		(TestCallerRef)&testcaller,\
	}

/* Adds a test set with description to the fixture of test sets.
See UNITTEST_TESTSET_FIXTURES() */
#define skipTestSet(testcaller)\
	{\
		1,\
		(TestCallerRef)&testcaller,\
	}

/* Adds a test set with description to the fixture of test sets.
See UNITTEST_TESTSET_FIXTURES() */
#define disabledTestSet(testcaller)\
	{\
		0,\
		(TestCallerRef)&testcaller,\
	}

/* Defines the test set list handling structure*/
#define UNTITTEST_TESTSET_HANDLER() \
TestSetList setList = {\
	sizeof(utTestSets) / sizeof(TestSetActive), \
	0, \
	(TestSetActive*)&utTestSets\
	}

#endif/*__HELPERMACRO_H__*/
```

### TestCase.h
```c
/*
* Author: 		B+R
* Contents of this file are modified and extended
*/

/*
 * COPYRIGHT AND PERMISSION NOTICE
 *
 * Copyright (c) 2003 Embedded Unit Project
 *
 * All rights reserved.
 *
 * Permission is hereby granted, free of charge, to any person obtaining
 * a copy of this software and associated documentation files (the
 * "Software"), to deal in the Software without restriction, including
 * without limitation the rights to use, copy, modify, merge, publish,
 * distribute, and/or sell copies of the Software, and to permit persons
 * to whom the Software is furnished to do so, provided that the above
 * copyright notice(s) and this permission notice appear in all copies
 * of the Software and that both the above copyright notice(s) and this
 * permission notice appear in supporting documentation.
 *
 * THE SOFTWARE IS PROVIDED "AS IS", WITHOUT WARRANTY OF ANY KIND,
 * EXPRESS OR IMPLIED, INCLUDING BUT NOT LIMITED TO THE WARRANTIES OF
 * MERCHANTABILITY, FITNESS FOR A PARTICULAR PURPOSE AND NONINFRINGEMENT
 * OF THIRD PARTY RIGHTS. IN NO EVENT SHALL THE COPYRIGHT HOLDER OR
 * HOLDERS INCLUDED IN THIS NOTICE BE LIABLE FOR ANY CLAIM, OR ANY
 * SPECIAL INDIRECT OR CONSEQUENTIAL DAMAGES, OR ANY DAMAGES WHATSOEVER
 * RESULTING FROM LOSS OF USE, DATA OR PROFITS, WHETHER IN AN ACTION OF
 * CONTRACT, NEGLIGENCE OR OTHER TORTIOUS ACTION, ARISING OUT OF OR IN
 * CONNECTION WITH THE USE OR PERFORMANCE OF THIS SOFTWARE.
 *
 * Except as contained in this notice, the name of a copyright holder
 * shall not be used in advertising or otherwise to promote the sale,
 * use or other dealings in this Software without prior written
 * authorization of the copyright holder.
 *
 * $Id: TestCase.h,v 1.7 2004/02/10 16:19:29 arms22 Exp $
 */
#ifndef	__TESTCASE_H__
#define	__TESTCASE_H__

typedef struct __TestCase	TestCase;
typedef struct __TestCase	*TestCaseRef;/*compatible embUnit1.0*/

struct __TestCase
{
	TestImplement 	*isa;
	const char 		*name;
	unsigned long	mode;
	testStateEnum 	state;
	char 			abort;
	testStatusEnum (*setUp)(void);
	testStatusEnum (*tearDown)(void);
	testStatusEnum (*runTest)(void);

};

extern const TestImplement TestCaseImplement;

#define new_TestCase(name,setUp,tearDown,runTest)\
	{\
		(TestImplement*)&TestCaseImplement,\
		name,\
		0, \
		stateStart,\
		0,\
		setUp,\
		tearDown,\
		runTest\
	}

#endif/*__TESTCASE_H__*/
```

### UtMgr.typ
```iecst
(********************************************************************
 * COPYRIGHT -- Bernecker + Rainer
 ********************************************************************
 * Library: UtMgr
 * File: UtMgr.typ
 * Author: B+R
 ********************************************************************
 * Data types of library UtMgr
 ********************************************************************)

TYPE
	UtMgrLocationType : 	STRUCT  (*Provides location information as passed by a assert*)
		TestSetName : UDINT; (*&STRING Name of current Test Set*)
		TestCaseName : UDINT; (*&STRING Name of current Test Case*)
		Line : UDINT; (*Line number (utMgrTEST_TYPE_C)*)
		Location : UDINT; (*&STRING Location information *)
		File : UDINT; (*&STRING File name*)
	END_STRUCT;
	UtMgrInformationalType : 	STRUCT  (*Informational Data, will be reset before test run is active*)
		TestCasesSinceActiveCounter : UDINT; (*Counts executed test cases (increments at the beginning of a test case)*)
		FailedAssertCounter : UDINT; (*Counts total failed asserts since start of testsuite execution *)
		PassedAssertCounter : UDINT; (*Counts total passed asserts since start of testsuite execution *)
		InformationalMessageCounter : UDINT; (*Counts total informational messages since start of testsuite execution *)
		LastKnownPassedLocation : UtMgrLocationType; (*Provides information about last known location (as reported in a test assert)*)
	END_STRUCT;
	UtMgrTestTypeEnum :
		( (*Defines Implementation of  UtMgrTestSuite*)
		utMgrTEST_TYPE_NONE := 0, (*Invalid value*)
		utMgrTEST_TYPE_C := 10, (*Test Suite uses the static library UnitTest *)
		utMgrTEST_TYPE_OTHER := 20 (*Reserved*)
		);
	UtMgrTestPhaseBasicHelperEnum :
		( (*Internal status of test execution*)
		utMgrTEST_PHASE_IDLE := 0, (*No tests running*)
		utMgrTEST_PHASE_RUNNING := 5, (*Executing Test Sets*)
		utMgrTEST_PHASE_DONE := 10 (*Done executing Test Sets*)
		);
	UtMgrUnitTestRunnerHelperType : 	STRUCT  (*Internal*)
		TestSets : UDINT; (*Pointer to the array of Test Sets*)
		TestSetCount : UINT; (*Number of entries in array*)
		CurrentPhase : UtMgrTestPhaseBasicHelperEnum; (*Status of internal test execution*)
		CurrentTestSet : UINT; (*Index of current active Test Set*)
	END_STRUCT;
	UtMgrSuiteInternalType : 	STRUCT  (*Internal*)
		State : DINT; (*Internal*)
		Handle : UDINT; (*Internal*)
		List : ARRAY[0..29]OF UDINT; (*Internal*)
		LibInst : UDINT; (*Internal*)
		TestHelper : UtMgrUnitTestRunnerHelperType; (*Internal*)
	END_STRUCT;
END_TYPE
```

### UtMgr.var
```iecst
(********************************************************************
 * COPYRIGHT -- Bernecker + Rainer
 ********************************************************************
 * Library: UtMgr
 * File: UtMgr.var
 * Author: B+R
 ********************************************************************
 * Constants of library UtMgr
 ********************************************************************)
VAR CONSTANT
	utERR_GENERAL : DINT := -1057750784; (*General error, see help*)
	utMgrERR_INVALID_PARAM : DINT := -1057750783; (*Check parameters*)
	utMgrERR_TOO_MANY_TESTS : DINT := -1057750782; (*Too many UtMgrTestSuites enabled, disable unused instances*)
END_VAR
```

- THIRDPARTYLICENSEREADME (not shown)

- ReplicateTest.py (not shown)

- Program Logical/UnitTest/Tests/BeltTests (ANSIC) (no source held here)

### Program Logical/UnitTest/Tests/BlockTests

#### BlockTests.var
```iecst
(********************************************************************
 * COPYRIGHT -- Bernecker + Rainer
 ********************************************************************
 * Program: BlockTests
 * Author: Jorge Murria
 ********************************************************************
 * Local variables of program BlockTests
 * General variables - do not change
 ********************************************************************)
(*Describe the test*)
VAR
	Testsuite : UtMgrTestSuite := (Name:='BlockTests',Description:='Description of the Tests',Type:=utMgrTEST_TYPE_C,MetaInformation:='Some Meta Information can be added here');
END_VAR
(*Variables used in the tests*)
```

#### autoGeneratedFile.c
```c
/*
B+R UnitTest: This is generated code.
Do not edit! Do not move!
Description: UnitTest Testprogramm infrastructure (List of TestSets).
LastUpdated: 2020-05-18 14:29:28Z
By B+R UnitTest Helper Version: 2.0.1.59
*/
#include "UnitTest.h"

UNITTEST_TESTSET_DECLARATION  BlockTests;

UNITTEST_TESTSET_FIXTURES(utTestSets)
{
	new_TestSet(BlockTests),
};
UNTITTEST_TESTSET_HANDLER();
```
